FUNCTION_BLOCK "V90_Servo"
VAR
  Servo_380A1 : "fbV90Ctrl";
  Servo_381A1 : "fbV90Ctrl";
  Servo_382A1 : "fbV90Ctrl";
  Servo_383A1 : "fbV90Ctrl";
  Servo1 : "SevroStart&PosCheck";
  Servo2 : "SevroStart&PosCheck";
  Servo3 : "SevroStart&PosCheck";
  Servo4 : "SevroStart&PosCheck";
  Servo2SafetyPos : DInt;
  Servo4SafetyPos : DInt;
  IEC_Timer_0_Instance : TON_TIME;
  P : Array[0..10] of Bool;
END_VAR
VAR_TEMP
  Sevro1ActPos : Real;
  Sevro1StartList : Bool;
  Sevro2ActPos : Real;
  Sevro2StartList : Bool;
  Sevro3ActPos : Real;
  Sevro3StartList : Bool;
  Sevro4ActPos : Real;
  Sevro4StartList : Bool;
END_VAR
BEGIN
  // Původní jazyk: LAD
  // Zdroj XML: EXPORT/Program blocks/OP010/10_Device/25_V90/V90_Servo.xml
  // --- Rekonstruovaný StructuredText (best-effort) ---
  // Network 1
  IF ..Station_Sys.Status.Run THEN
       ..[]. := ..[]. :=(..[]..*);
       ..[]. := ..[]. := ..[]..;

       ..[]. := ..[]. := (..[]..*);
      ..[]. := ..[]. := ..[]..;

      ..[]. := ..[]. := (..[]..*);
      ..[]. := ..[]. := ..[]..;

      ..[]. := ..[]. := (..[]..*);
      ..[]. := ..[]. := ..[]..;

      ..[]. := ..[]. := (..[]..*);
      ..[]. := ..[]. := ..[]..;

      ..[]. := ..[]. := (..[]..*);
      ..[]. := ..[]. := ..[]..;

      ..[]. := ..[]. := (..[]..*);
      ..[]. := ..[]. := ..[]..;

      ..[]. := ..[]. := (..[]..*);
      ..[]. := ..[]. := ..[]..;

      ..[]. := ..[]. := (..[]..*);
      ..[]. := ..[]. := ..[]..;

  END_IF;
  // Network 2
  IF ..Station_Sys.Status.Run THEN
       ..[]. := ..[]. := (..[]..*);
      ..[]. := ..[]. := ..[]..;

      ..[]. := ..[]. := (..[]..*);
      ..[]. := ..[]. := ..[]..;

      ..[]. := ..[]. := (..[]..*);
      ..[]. := ..[]. := ..[]..;

      ..[]. := ..[]. := (..[]..*);
      ..[]. := ..[]. := ..[]..;

      ..[]. := ..[]. := (..[]..*);
      ..[]. := ..[]. := ..[]..;

      ..[]. := ..[]. := (..[]..*);
      ..[]. := ..[]. := ..[]..;

      ..[]. := ..[]. := (..[]..*);
      ..[]. := ..[]. := ..[]..;

      ..[]. := ..[]. := (..[]..*);
      ..[]. := ..[]. := ..[]..;

      ..[]. := ..[]. := (..[]..*);
      ..[]. := ..[]. := ..[]..;

      ..[]. := ..[]. := (..[]..*);
      ..[]. := ..[]. := ..[]..;
  END_IF;
  // Network 3
  IF ..Station_Sys.Status.Run THEN
       ..[]. := ..[]. := (..[]..*);
       ..[]. := ..[]. := ..[]..;

       ..[]. := ..[]. := (..[]..*);
       ..[]. := ..[]. := ..[]..;

       ..[]. := ..[]. := (..[]..*);
       ..[]. := ..[]. := ..[]..;

       ..[]. := ..[]. := (..[]..*);
       ..[]. := ..[]. := ..[]..;

       ..[]. := ..[]. := (..[]..*);
       ..[]. := ..[]. := ..[]..;

       ..[]. := ..[]. := (..[]..*);
       ..[]. := ..[]. := ..[]..;

       ..[]. := ..[]. := (..[]..*);
       ..[]. := ..[]. := ..[]..;

       ..[]. := ..[]. := (..[]..*);
       ..[]. := ..[]. := ..[]..;

       ..[]. := ..[]. := (..[]..*);
       ..[]. := ..[]. := ..[]..;

       ..[]. := ..[]. := (..[]..*);
       ..[]. := ..[]. := ..[]..;
  END_IF;
  // Network 4
  IF ..Station_Sys.Status.Run THEN
      ..[]. := ..[]. := (..[]..*);
      ..[]. := ..[]. := ..[]..;

      ..[]. := ..[]. := (..[]..*);
      ..[]. := ..[]. := ..[]..;

      ..[]. := ..[]. := (..[]..*);
      ..[]. := ..[]. := ..[]..;

      ..[]. := ..[]. := (..[]..*);
      ..[]. := ..[]. := ..[]..;

      ..[]. := ..[]. := (..[]..*);
      ..[]. := ..[]. := ..[]..;

      ..[]. := ..[]. := (..[]..*);
      ..[]. := ..[]. := ..[]..;

      ..[]. := ..[]. := (..[]..*);
      ..[]. := ..[]. := ..[]..;

      ..[]. := ..[]. := (..[]..*);
      ..[]. := ..[]. := ..[]..;

      ..[]. := ..[]. := (..[]..*);
      ..[]. := ..[]. := ..[]..;

      ..[]. := ..[]. := (..[]..*);
      ..[]. := ..[]. := ..[]..;
  END_IF;
  // Network 5
  FOR .[]. :=  TO  BY  DO
      .[]..[.[].]. := ..[.[].].;
      .[]..[.[].]. := ..[.[].].;

      .[]..[.[].]. := ..[.[].].;
      .[]..[.[].]. := ..[.[].].;

      .[]..[.[].]. := ..[.[].].;
      .[]..[.[].]. := ..[.[].].;

      .[]..[.[].]. := ..[.[].].;
      .[]..[.[].]. := ..[.[].].;

  END_FOR;


  ( :=   ..ServoV90_A1.Out.oHomeRef,
                             := ,
                             := ..Station_Sys.Cmd.Reset,
                            :=..ServoV90_A1.In.iInterlock,
                             :=..ServoV90_A1.Out.oActPosition,
                             := ,
                             := ,
                             := ,
                            :=.[].,
                             => #Sevro1StartList,
                             := .[].,
                             := .[].);

  IF .[]. =  THEN
     .[].:=  ;
  END_IF;






                 ..ServoV90_A1.Auto.Index := .[].;


                  ..ServoV90_A1.In.iAutoStart := #Sevro1StartList;




  ( := ..ServoV90_A2.Out.oHomeRef,
             := ,
             := ..Station_Sys.Cmd.Reset,
             := ..ServoV90_A2.In.iInterlock,
             := ..ServoV90_A2.Out.oActPosition,
             := ,
             := ,
             := ,
             := .[].,
             => #Sevro2StartList,
             := .[].,
             := .[].);
  IF .[]. =  THEN
      .[]. := ;
  END_IF;




  ..ServoV90_A2.Auto.Index := .[].;

  ..ServoV90_A2.In.iAutoStart := #Sevro2StartList;




  ( := ..ServoV90_A3.Out.oHomeRef,
             := ,
             := ..Station_Sys.Cmd.Reset,
             := ..ServoV90_A3.In.iInterlock,
             := ..ServoV90_A3.Out.oActPosition,
             := ,
             := ,
             := ,
             := .[].,
             => #Sevro3StartList,
             := .[].,
             := .[].);
  IF .[]. =  THEN
      .[]. := ;
  END_IF;




  ..ServoV90_A3.Auto.Index := .[].;

  ..ServoV90_A3.In.iAutoStart := #Sevro3StartList;


  ( := ..ServoV90_A4.Out.oHomeRef,
             := ,
             := ..Station_Sys.Cmd.Reset,
             := ..ServoV90_A4.In.iInterlock,
             := ..ServoV90_A4.Out.oActPosition,
             := ,
             := ,
             := ,
             := .[].,
             => #Sevro4StartList,
             := .[].,
             := .[].);
  IF .[]. =  THEN
      .[]. := ;
  END_IF;




  ..ServoV90_A4.Auto.Index := .[].;

  ..ServoV90_A4.In.iAutoStart := #Sevro4StartList;
  // Network 6
  IF FirstScan THEN
      ..ServoV90_A1.IO.ioManEnale := ;
      ..ServoV90_A2.IO.ioManEnale := ;
      ..ServoV90_A3.IO.ioManEnale := ;
      ..ServoV90_A4.IO.ioManEnale := ;
  END_IF;
  // --- LAD/FBD → SCL (orientační převod, jen pro revizi) ---
  // Network 1
  // --- Poznámky / omezení převodu ---
  // Síť obsahuje nepodporované prvky (ponecháno jen jako komentář): O(1)
  // RCoil UId=27: nelze určit podmínku (vstupní síť).
  // Network 2
  // --- Poznámky / omezení převodu ---
  // Síť obsahuje nepodporované prvky (ponecháno jen jako komentář): Move(1)
  // Network 3
  ServoV90_A1.Interlock.Case1 := Station_Sys.Status.Run;
  ServoV90_A1.Interlock.Case2 := Station_Sys.Status.Run;
  ServoV90_A1.In.iInterlock := ((Station_Sys.Status.Run AND ServoV90_A1.Interlock.Case1) AND ServoV90_A1.Interlock.Case2);
  // Network 4
  ServoV90_A1.IO.ioAutoEnale := (((AlwaysTRUE AND Station_Sys.Auto.Mode) AND Station_Sys.Status.Run) AND iALightCurtain_1);
  IF (AlwaysTRUE AND NOT iALightCurtain_1) THEN ServoV90_A1.IO.ioManEnale := FALSE; END_IF;
  // --- Poznámky / omezení převodu ---
  // Síť obsahuje nepodporované prvky (ponecháno jen jako komentář): PBox(2), Move(1)
  // SCoil UId=46: nelze určit podmínku (vstupní síť).
  // SCoil UId=50: nelze určit podmínku (vstupní síť).
  // Network 5
  // Network 6
  // --- Poznámky / omezení převodu ---
  // Síť obsahuje nepodporované prvky (ponecháno jen jako komentář): O(1)
  // RCoil UId=27: nelze určit podmínku (vstupní síť).
  // Network 7
  // --- Poznámky / omezení převodu ---
  // Síť obsahuje nepodporované prvky (ponecháno jen jako komentář): Move(1)
  // Network 8
  ServoV90_A2.Interlock.Case1 := Station_Sys.Status.Run;
  ServoV90_A2.Interlock.Case2 := Station_Sys.Status.Run;
  ServoV90_A2.In.iInterlock := ((Station_Sys.Status.Run AND ServoV90_A2.Interlock.Case1) AND ServoV90_A2.Interlock.Case2);
  // Network 9
  ServoV90_A2.IO.ioAutoEnale := ((AlwaysTRUE AND Station_Sys.Status.Run) AND Station_Sys.Auto.Mode);
  // --- Poznámky / omezení převodu ---
  // Síť obsahuje nepodporované prvky (ponecháno jen jako komentář): PBox(2), Move(1)
  // SCoil UId=40: nelze určit podmínku (vstupní síť).
  // SCoil UId=44: nelze určit podmínku (vstupní síť).
  // Network 10
  // Network 11
  // --- Poznámky / omezení převodu ---
  // Síť obsahuje nepodporované prvky (ponecháno jen jako komentář): O(1)
  // RCoil UId=27: nelze určit podmínku (vstupní síť).
  // Network 12
  // --- Poznámky / omezení převodu ---
  // Síť obsahuje nepodporované prvky (ponecháno jen jako komentář): Move(1)
  // Network 13
  ServoV90_A3.Interlock.Case1 := Station_Sys.Status.Run;
  ServoV90_A3.Interlock.Case2 := Station_Sys.Status.Run;
  ServoV90_A3.In.iInterlock := ((Station_Sys.Status.Run AND ServoV90_A3.Interlock.Case1) AND ServoV90_A3.Interlock.Case2);
  // Network 14
  ServoV90_A3.IO.ioAutoEnale := ((AlwaysTRUE AND Station_Sys.Status.Run) AND Station_Sys.Auto.Mode);
  // --- Poznámky / omezení převodu ---
  // Síť obsahuje nepodporované prvky (ponecháno jen jako komentář): PBox(2), Move(1)
  // SCoil UId=39: nelze určit podmínku (vstupní síť).
  // SCoil UId=42: nelze určit podmínku (vstupní síť).
  // Network 15
  // --- Poznámky / omezení převodu ---
  // Síť obsahuje nepodporované prvky (ponecháno jen jako komentář): Eq(2), O(1)
  // Network 16
  IF ServoV90_DeviceCtl.V90Servo THEN ServoV90_DeviceCtl.V90Servo := FALSE; END_IF;
  // Network 17
  // --- Poznámky / omezení převodu ---
  // Síť obsahuje nepodporované prvky (ponecháno jen jako komentář): O(1)
  // RCoil UId=27: nelze určit podmínku (vstupní síť).
  // Network 18
  // --- Poznámky / omezení převodu ---
  // Síť obsahuje nepodporované prvky (ponecháno jen jako komentář): Move(1)
  // Network 19
  ServoV90_A4.Interlock.Case1 := Station_Sys.Status.Run;
  ServoV90_A4.Interlock.Case2 := Station_Sys.Status.Run;
  ServoV90_A4.In.iInterlock := ((Station_Sys.Status.Run AND ServoV90_A4.Interlock.Case1) AND ServoV90_A4.Interlock.Case2);
  // Network 20
  ServoV90_A4.IO.ioAutoEnale := (((AlwaysTRUE AND Station_Sys.Status.Run) AND Station_Sys.Auto.Mode) AND iALightCurtain_2);
  IF (AlwaysTRUE AND NOT iALightCurtain_2) THEN ServoV90_A4.IO.ioManEnale := FALSE; END_IF;
  // --- Poznámky / omezení převodu ---
  // Síť obsahuje nepodporované prvky (ponecháno jen jako komentář): PBox(2), Move(1)
  // SCoil UId=46: nelze určit podmínku (vstupní síť).
  // SCoil UId=50: nelze určit podmínku (vstupní síť).
  // Network 21
END_FUNCTION_BLOCK
